// TIA Portal V19 export
FUNCTION "TOTAL STOP" : Void   // FC42, STL
TITLE = TOTAL STOP ASEPTIC TANK
{ S7_Optimized_Access := 'TRUE' }
NAME : TSTOPTNK
// ****** REVISION HISTORY :
// 
// VERSION DATE       BY  DESCRIPTION
// --------------------------------------------------------------------------
// 00.00               ORIGINAL FUNCTION BLOCK
// 
// 00.01 10/12 1997   OPA
//       FOLLOWING INSTRUCTIONS HAVE BEEN ADDED IN NETWORK 1
//       R     "S.T.01.REQUEST LYE"   "M242.0"     // STOP REQUESTING DETERGENT
//       R     "S.T.01.REQUEST ACID"  "M242.1"     // STOP REQUESTING DETERGENT
//       WITHOUT THESE TWO INSTRUCTIONS, DETERGENT PUMPS (LYE/ACID) COULD
//       CONTINUE DOSING AFTER STOP.
// stored: AutoNumber false
BEGIN

NETWORK
TITLE = TOTAL STOP ASEPTIC TANK
// Comment
      AN    "S0 TOTAL STOP TANK";
      R     "S1 TOTAL STOP TANK";
      R     "S2 TOTAL STOP TANK";
      BEC;
      A     "S1 TOTAL STOP TANK";
      JC    M001;
      S     "MY0112";
//      R     "MY0113"
      S     "MY0113";  // BUG 300699 on reguest
      R     "MY0147";
//      S     "MY0118"
      R     "MY0118";  // BUG 300699 on request
      R     "MY0116";  // BUG 300699 on request
      S     "MY0114";  // BUG 300699 on request
      S     "MY0111";
      R     "AutoPT0167/IP0149";
      R     "ManPT0167/IP0149";
      R     "AutoTT0172/IP0157";
      R     "ManTT0172/IP0157";
      R     "MM0139";
      R     "MY0158";
//     R     "MM01.30"
      R     "SPIN 01.30 PRESTERILI";
      R     "PULSE 01.18 PRESTERILI";
      R     "CONTROL CIP TANK";
      R     "PULSE 01.08 CIP";
      R     "SPIN 01.30 CIP";
      R     "PULSE 01.13 CIP";
      R     "MY0136";
      R     "MY0137";
      R     "MY0135";
      R     "MY0103";
      R     "MY0104";
      R     "MY0108";
      R     "MY0124";
      R     "MY0144";
      S     "TIM17";
      R     "S.T.01.REQUEST LYE";  // STOP REQUESTING DETERGENT
      R     "S.T.01.REQUEST ACID";  // STOP REQUESTING DETERGENT
      R     "T 27 WATER 1";
      R     "T 28 DOSING LYE";
      R     "T 29 LYE CIRCULATION";
      R     "T 30 WATER 2";
      R     "T 31 DOSING ACID";
      R     "T 32 ACID CIRCULATION";
      R     "T 33 WATER 3";
      R     "T 34 BLOW OUT CIP";
      R     "MY0901";
      R     "MY0904";
      R     "MY0906";
      R     "MY0907";
      S     "S1 TOTAL STOP TANK";
      BEU;
M001: NOP   0;

NETWORK
TITLE = 
// Comment
      A     "S2 TOTAL STOP TANK";
      JC    c001;
      A     "T 17 BLOW OUT STOP";
      BEC;
      R     "S0 TOTAL STOP TANK";
      BEU;
c001: NOP   0;
END_FUNCTION
